{attribute 'pack_mode' := '2'}
TYPE ST_XPU_STATE :
STRUCT
  Init            : E_XPU_INIT;
  State           : E_XPU_STATE;
  Check           : E_XPU_CHECK;  // cyclic check result
  DcLink          : BIT;          // power all motor modules is ON
END_STRUCT
END_TYPE

(* stored: Version 1.1.0.1
   DUT ST_XPU_STATE: Id {d88dffc7-d64d-4f49-8f55-bbe6ccdbd195} *)
